Staubli VAL3: _tPLC.pgx

public program _tPLC()
  local bool l_bContinue
  local bool l_bStopStatus
begin
  while true

    io:dOutIsReady=(bIsHome and bIsRemote and !bIsEstop and !bRobotErr and !bCycle)
    if io:dOutIsReady==true
      bIsReady=true
    endIf

    //远程自动上电
    if io:dInStart==true
      if taskStatus("cycle")==-1 and bIsReady==true
        bCycle=true
        call PowerOn(l_bContinue)
        if l_bContinue==true
          taskCreate "cycle",100,_tcycle()
          wait(taskStatus("cycle")==1)
        else
          bCycle=false
        endIf
      endIf
      endIf

    if bCycle==true
      call isStopped(l_bStopStatus)
    endIf

  endWhile
end
